% RSLogix 500 project Retentive Timer Motor Control.RSS, saved by version 8.30.00.16 %
PROJECT "UNTITLED"    % processor: Bul.1763 MicroLogix 1100 Series B %

PROGRAM FILES
  LAD 2   4 rungs

DATA FILES
  O0 OUTPUT  4 elements
  I1 INPUT  6 elements
  S2 STATUS  66 elements
  B3 BINARY  1 elements
  T4 TIMER  1 elements
  C5 COUNTER  1 elements
  R6 CONTROL  1 elements
  N7 INTEGER  1 elements
  F8 FLOAT  1 elements

LADDER 2
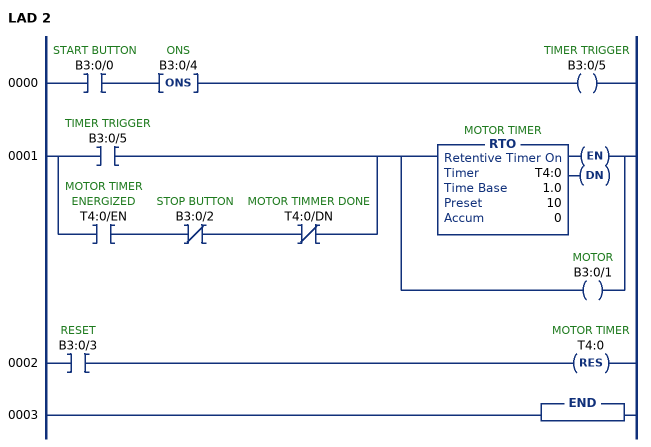
% Rung: 0 %
SOR XIC B3:0/0 ONS B3:0/4 OTE B3:0/5 EOR
%   B3:0/0  "START BUTTON" %
%   B3:0/4  "ONS" %
%   B3:0/5  "TIMER TRIGGER" %
% Rung: 1 %
SOR BST XIC B3:0/5 NXB XIC T4:0/EN XIO B3:0/2 XIO T4:0/DN BND BST RTO T4:0 1.0 10 0 NXB OTE B3:0/1 BND EOR
%   B3:0/5  "TIMER TRIGGER" %
%   T4:0/EN  "MOTOR TIMER ENERGIZED" %
%   B3:0/2  "STOP BUTTON" %
%   T4:0/DN  "MOTOR TIMMER DONE" %
%   T4:0  "MOTOR TIMER" %
%   B3:0/1  "MOTOR" %
% Rung: 2 %
SOR XIC B3:0/3 RES T4:0 EOR
%   B3:0/3  "RESET" %
%   T4:0  "MOTOR TIMER" %
% Rung: 3 %
SOR END EOR

DATA TABLE (non-zero values as saved)
DATA T4
% .PRE .ACC %
% T4:0 % 10 0
